TYPE ST_PNOZRawIn :
STRUCT
    aSafetyFunction : ARRAY[1..GVL_SafetyIO.UPPER_BOUND_SF_INPUT] OF ST_SafetyFunctionIn;
END_STRUCT
END_TYPE

(* stored: Version 1.1.0.1
   DUT ST_PNOZRawIn: Id {40acf446-3183-47fb-8d3f-0dd7b158d9d4} *)
